{attribute 'GeneratedUsingTerminal: EPP1342-0001-0017'}
{attribute addProperty BoxType "EPP1342-0001-0017"}
{attribute addProperty Id "A_0025_EPP1518_0002_0016EPP1518_1B7BBD8659A_0026_EPP1518_0002_0017EPP1518_1B7BBD8659A_0027_EPP1809_0021_0016EPP1809_FD7895E220A_0028_EPP1809_0022_0016EPP1809_FD7895E220A_0029_EPP1819_0021_0016EPP1819_FD7895E220A_0030_EPP1819_0022_0016EPP1819_FD7895E220A_0031_EPP1816_0003_0016EPP1816_9F97CFEF32A_0032_EPP1816_0008_0016EPP1816_6247929530A_0033_EPP1816_0008_0017EPP1816_6247929530A_0034_EPP1816_0008_0018EPP1816_9F97CFEF32A_0035_EPP1816_3008_0016EPP1816_4FA00BC356"}
{attribute addProperty CRC "560439694"}
{attribute addProperty Size "378"}
TYPE A_0024_EPP1342_0001_0017_2167A18E EXTENDS EPP1342_AB5A9467 :
STRUCT
	{attribute addProperty Name "A_0025_EPP1518_0002_0016"}
	{attribute addProperty PreviousPort "A_0024(EPP1342-0001-0017) : D"}
	A_0025_EPP1518_0002_0016 : EPP1518_1B7BBD86;
	{attribute addProperty Name "A_0026_EPP1518_0002_0017"}
	{attribute addProperty PreviousPort "A_0025(EPP1518-0002-0016) : B"}
	A_0026_EPP1518_0002_0017 : EPP1518_1B7BBD86;
	{attribute addProperty Name "A_0027_EPP1809_0021_0016"}
	{attribute addProperty PreviousPort "A_0026(EPP1518-0002-0017) : B"}
	A_0027_EPP1809_0021_0016 : EPP1809_FD7895E2;
	{attribute addProperty Name "A_0028_EPP1809_0022_0016"}
	{attribute addProperty PreviousPort "A_0027(EPP1809-0021-0016) : B"}
	A_0028_EPP1809_0022_0016 : EPP1809_FD7895E2;
	{attribute addProperty Name "A_0029_EPP1819_0021_0016"}
	{attribute addProperty PreviousPort "A_0028(EPP1809-0022-0016) : B"}
	A_0029_EPP1819_0021_0016 : EPP1819_FD7895E2;
	{attribute addProperty Name "A_0030_EPP1819_0022_0016"}
	{attribute addProperty PreviousPort "A_0029(EPP1819-0021-0016) : B"}
	A_0030_EPP1819_0022_0016 : EPP1819_FD7895E2;
	{attribute addProperty Name "A_0031_EPP1816_0003_0016"}
	{attribute addProperty PreviousPort "A_0030(EPP1819-0022-0016) : B"}
	A_0031_EPP1816_0003_0016 : EPP1816_9F97CFEF;
	{attribute addProperty Name "A_0032_EPP1816_0008_0016"}
	{attribute addProperty PreviousPort "A_0031(EPP1816-0003-0016) : B"}
	A_0032_EPP1816_0008_0016 : EPP1816_62479295;
	{attribute addProperty Name "A_0033_EPP1816_0008_0017"}
	{attribute addProperty PreviousPort "A_0032(EPP1816-0008-0016) : B"}
	A_0033_EPP1816_0008_0017 : EPP1816_62479295;
	{attribute addProperty Name "A_0034_EPP1816_0008_0018"}
	{attribute addProperty PreviousPort "A_0033(EPP1816-0008-0017) : B"}
	A_0034_EPP1816_0008_0018 : EPP1816_9F97CFEF;
	{attribute addProperty Name "A_0035_EPP1816_3008_0016"}
	{attribute addProperty PreviousPort "A_0034(EPP1816-0008-0018) : B"}
	A_0035_EPP1816_3008_0016 : EPP1816_4FA00BC3;
END_STRUCT
END_TYPE

(* stored: Version 1.2.0.0, ProductVersion 3.1.4024.9
   DUT A_0024_EPP1342_0001_0017_2167A18E: Id {450def71-b537-4061-b862-dc2b908368ff} *)
